FUNCTION_BLOCK E_SWITCH
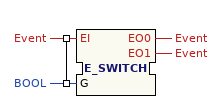
  EVENT_INPUT
    EI WITH G;
  END_EVENT
  EVENT_OUTPUT
    EO0;
    EO1;
  END_EVENT
  VAR_INPUT
    G : BOOL;
  END_VAR
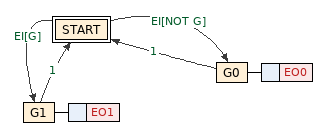
  EC_STATES
    START;
    G0 : -> EO0;
    G1 : -> EO1;
  END_STATES
  EC_TRANSITIONS
    G0 TO START := 1;
    G1 TO START := 1;
    START TO G0 := EI[NOT G];
    START TO G1 := EI[G];
  END_TRANSITIONS
END_FUNCTION_BLOCK
